// TwinCAT 3 PLC project Singleton1
// ProgramVersion: 3.1.4023.0
// libraries:
//   Tc2_Standard, * (Beckhoff Automation GmbH)
//   Tc2_System, * (Beckhoff Automation GmbH)
//   Tc3_Module, * (Beckhoff Automation GmbH)
//   VisuSymbols,3.5.10.0,System
// project tree:
//   / Class Diagram_2.TcCD (not stored), E_Color.TcDUT (not stored), GlobalTextList.TcGTLO, PlcTask.TcTTO (not stored), PLC_PRG.TcPOU, ProxyToSingleton.TcPOU, Proxy_Interface.TcIO (not stored), RealSingleton.TcPOU, Visualization Manager.TcVMO (not stored)
//   POUs/ MAIN.TcPOU (not stored)
//   VISUs/ Visualization.TcVIS
// real-time tasks:
//   TASK PlcTask: cycle T#10ms, priority 20, ADS port 350

// ---- PLC_PRG.TcPOU
PROGRAM PLC_PRG
VAR
	///Blue, highly opaque
	dwBlue: DWORD := 16#FF0000FF;
	///Green, highly opaque
	dwGreen: DWORD := 16#FF00FF00;
	///Yellow, highly opaque
	dwYellow: DWORD := 16#FFFFFFF0;
	///Creates 3 instances of the ProxyToSingleton class
	instance1: ProxyToSingleton;
	instance2: ProxyToSingleton;
	instance3: ProxyToSingleton;
	
	eInstance1 : E_Color;
	eInstance2 : E_Color;
	eInstance3 : E_Color;
	
END_VAR

//*************************************************************************************************************************************************************
//The PLC_PRG handles the instanciation of the possible background colours and the ProxyToSingleton instances in order to be used by the Visualization element.
//The viasualization element (The client) handles the request for background change on the RealSingleton object through the ProxyToSinlgeton instances.
//These request are first processed by the ProxyToSingleton object and then passed to the one and only RealSingleton instance.
//The default background colour of the RealSingleton object is 'Blue' 
//*************************************************************************************************************************************************************
// spanish
//PLC_PRG maneja la instanciación de los posibles colores de fondo y las instancias de ProxyToSingleton para ser utilizados por el elemento de visualización.
//El elemento de visualización (el cliente) maneja la solicitud de cambio de fondo en el objeto RealSingleton a través de las instancias de ProxyToSinlgeton.
//Estas solicitudes son procesadas primero por el objeto ProxyToSingleton y luego pasadas a la única instancia de RealSingleton.
//El color de fondo predeterminado del objeto RealSingleton es 'Azul'
//*************************************************************************************************************************************************************

CASE eInstance1 OF
	E_Color.Blue:
		instance1.Set_Background(dwBlue);
		eInstance1:=E_Color.NoColor;
	E_Color.Green:
		instance1.Set_Background(dwGreen);
		eInstance1:=E_Color.NoColor;
	E_Color.Yellow:
		instance1.Set_Background(dwYellow);
		eInstance1:=E_Color.NoColor;
END_CASE

CASE eInstance2 OF
	E_Color.Blue:
		instance2.Set_Background(dwBlue);
		eInstance2:=E_Color.NoColor;	
	E_Color.Green:
		instance2.Set_Background(dwGreen);
		eInstance2:=E_Color.NoColor;	
	E_Color.Yellow:
		instance2.Set_Background(dwYellow);
		eInstance2:=E_Color.NoColor;	
END_CASE

CASE eInstance3 OF
	E_Color.Blue:
		instance3.Set_Background(dwBlue);
		eInstance3:=E_Color.NoColor;	
	E_Color.Green:
		instance3.Set_Background(dwGreen);
		eInstance3:=E_Color.NoColor;	
	E_Color.Yellow:
		instance3.Set_Background(dwYellow);
		eInstance3:=E_Color.NoColor;	
END_CASE

END_PROGRAM

// ---- ProxyToSingleton.TcPOU
///This class is called ProxyToSingleton because it works as a Proxy of the Singleton class. It handles the creation and instanciation of the 
/// RealSingleton class. Something like the proper static method GetInstance(); in any singleton pattern.
///So the ProxyToSingleton class has a static Singleton object as a field and whenever we instanciate a 
/// ProxyToSingleton object we will have the RealSingleton object as its static field .realSingleton^
{attribute 'enable_dynamic_creation' := ''}
FUNCTION_BLOCK ProxyToSingleton IMPLEMENTS Proxy_Interface
VAR_STAT
	///Boolean value to check if there is already a Singleton instance
	bFirstInstance: BOOL := FALSE;
	///Pointer to the first and only instance of the Singleton class
	realSingleton: POINTER TO RealSingleton;
END_VAR

METHOD fb_init
VAR_INPUT
	/// TRUE: the Retain-variables are initialized (reset warm / reset cold)
	bInitRetains: BOOL;
	/// TRUE  the instance will be copied to the copy-code afterward (online change)
	bInCopyCode: BOOL;
END_VAR
//THIS FUNCTION WORKS AS THE CONSTRUCTOR OF THE ProxyToSingleton CLASS
// It handles the creation of the only RealSingleton object. It uses the concept of lazy instanciation.

//If the static property .bFirstInstance is TRUE
IF THIS^.bFirstInstance = TRUE
	
THEN
		//There is already a Singleton object.
		//So we don't have to do anything, this new ProxyToSingleton object will already have the address of the 
		// RealSingleton object in its pointer .realSingleton
	
	ELSE	//If the static property .bFirstInstance is FALSE
	
		//There is not a Singleton object so the ProxyToSingleton object calling the constructor 
		// should create the RealSingleton object in its pointer field .realSingleton 
		//Then we change the status of the static variable bFirstInstance to TRUE and avoid overwriting the realSingleton address.
		//If the Singleton object is destroyed, .bFirstInstance should be set to FALSE again.
		THIS^.bFirstInstance := TRUE;
		
		//Reference the value of the first RealSingleton instance to the FakeSingleton object to save 
		// the address of the real Singleton instance.
		THIS^.realSingleton := __NEW(RealSingleton);
END_IF
END_METHOD

///Illustrative method of the pattern
METHOD Set_Background
VAR_INPUT
	///HEX value to be set as background color
	newBackground: DWORD;
END_VAR
//The ProxyToSingleton object handles the request and send the appropiate reques to the one and only RealSingleton instance
THIS^.realSingleton^.Set_Background(newBackground);
END_METHOD

END_FUNCTION_BLOCK

// ---- RealSingleton.TcPOU
///This class is called RealSingleton because it works as singleton.  
///As long as we only instanciate ProxyToSingleton objects, this class will work as a Singleton class should work.
///The global access point to this class is the field .realSingleton^ in every ProxyToSingleton object.
{attribute 'enable_dynamic_creation' := ''}
FUNCTION_BLOCK RealSingleton IMPLEMENTS Proxy_Interface
VAR
	///Illustrative field of the pattern to store the HEX value for the background colour
	backgroundColour: DWORD;
END_VAR

METHOD fb_init
VAR_INPUT
	/// TRUE: the Retain-variables are initialized (reset warm / reset cold)
	bInitRetains: BOOL;
	/// TRUE  the instance will be copied to the copy-code afterward (online change)
	bInCopyCode: BOOL;
END_VAR
//The default valur for the background is set
THIS^.Set_Background(PLC_PRG.dwBlue);
END_METHOD

///Illustrative method of the pattern
METHOD Set_Background
VAR_INPUT
	///HEX value to be set as background color
	newBackground: DWORD;
END_VAR
//Writes the backgroundColour field to the passed newBackground value
THIS^.backgroundColour := newBackground;
END_METHOD

END_FUNCTION_BLOCK

// ---- GlobalTextList.TcGTLO
TEXTLIST GlobalTextList
  630 = "//The PLC_PRG handles the instanciation of the possible background colours and the ProxyToSingleton instances in order to be used by the Visualization element.\n//The viasualization element (The client) handles the request for background change on the RealSingleton object through the ProxyToSinlgeton instances.\n//These request are first processed by the ProxyToSingleton object and then passed to the one and only RealSingleton instance.\n//The default background colour of the RealSingleton object is 'Blue' "
  622 = "//The PLC_PRG handles the instanciation of the possible background colours and the ProxyToSingleton instances in order to be used by the Visualization element.\n//The visualization element (The client) handles the request for background change on the RealSingleton object through the ProxyToSinlgeton instances.\n//These request are first processed by the ProxyToSingleton object and then passed to the one and only RealSingleton instance.\n//The default background colour of the RealSingleton object is 'Blue' "
  596 = 'instance1.realSingleton^.\nbackgroundColor'
  621 = 'instance1.Set_Background(HEX color)'
  436 = 'instance2.realSingleton^.\nbackgroundColor'
  534 = 'instance2.Set_Background(HEX color)'
  774 = 'instance3.realSingleton^.\nbackgroundColor'
  50 = 'instance3.Set_Background(HEX color)'
  430 = 'The PLC_PRG handles the instanciation of the possible background colours and the ProxyToSingleton instances in order to be used by the Visualization element.\n'
END_TEXTLIST

// ---- VISUs/Visualization.TcVIS
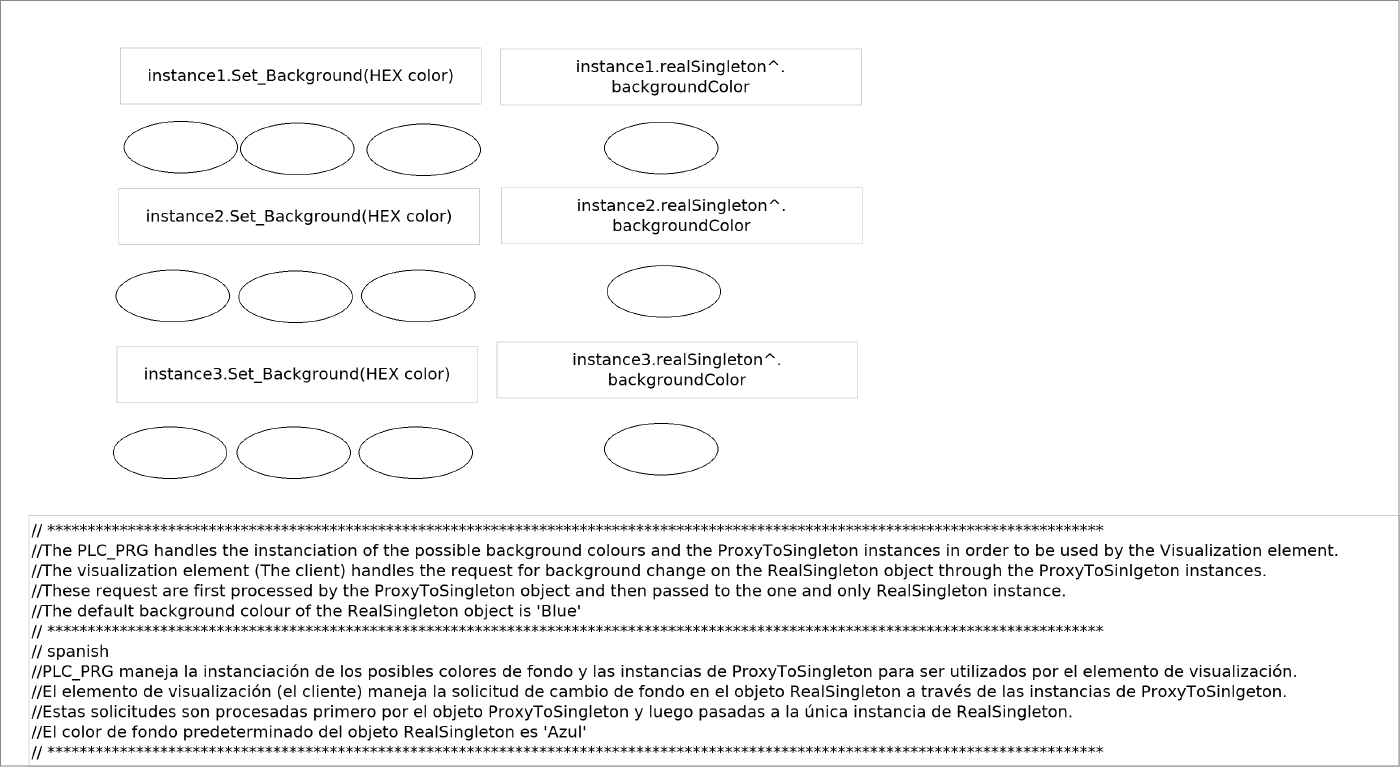
VISUALIZATION Visualization  // 1562x856
    Textfield (134,53 403x63), "instance1.Set_Background(HEX color)"
    Textfield (558,54 403x63), "instance1.realSingleton^. backgroundColor"
    Textfield (132,210 403x63), "instance2.Set_Background(HEX color)"
    Textfield (130,386 403x63), "instance3.Set_Background(HEX color)"
    Textfield (559,209 403x63), "instance2.realSingleton^. backgroundColor"
    Textfield (554,381 403x63), "instance3.realSingleton^. backgroundColor"
    Ellipse (138,135 127x58), colour variable: PLC_PRG.dwBlue
        OnMouseClick: execute {
            //PLC_PRG.instance1.Set_Background(newBackground:=PLC_PRG.dwBlue);
            PLC_PRG.eInstance1 := E_Color.Blue;
        }
    Ellipse (409,138 127x58), colour variable: PLC_PRG.dwYellow
        OnMouseClick: execute {
            //PLC_PRG.instance1.Set_Background(newBackground:=PLC_PRG.dwYellow);
            PLC_PRG.eInstance1 := E_Color.Yellow;
        }
    Ellipse (268,137 127x58), colour variable: PLC_PRG.dwGreen
        OnMouseClick: execute {
            //PLC_PRG.instance1.Set_Background(newBackground:=PLC_PRG.dwGreen);
            PLC_PRG.eInstance1 := E_Color.Green;
        }
    Ellipse (129,301 127x58), colour variable: PLC_PRG.dwBlue
        OnMouseClick: execute {
            //PLC_PRG.instance2.Set_Background(PLC_PRG.dwBlue);
            PLC_PRG.eInstance2 := E_Color.Blue;
        }
    Ellipse (403,301 127x58), colour variable: PLC_PRG.dwYellow
        OnMouseClick: execute {
            //PLC_PRG.instance2.Set_Background(PLC_PRG.dwYellow);
            PLC_PRG.eInstance2 := E_Color.Yellow;
        }
    Ellipse (266,302 127x58), colour variable: PLC_PRG.dwGreen
        OnMouseClick: execute {
            //PLC_PRG.instance2.Set_Background(PLC_PRG.dwGreen);
            PLC_PRG.eInstance2 := E_Color.Green;
        }
    Ellipse (126,476 127x58), colour variable: PLC_PRG.dwBlue
        OnMouseClick: execute {
            //PLC_PRG.instance3.Set_Background(PLC_PRG.dwBlue);
            PLC_PRG.eInstance3 := E_Color.Blue;
        }
    Ellipse (400,476 127x58), colour variable: PLC_PRG.dwYellow
        OnMouseClick: execute {
            //PLC_PRG.instance3.Set_Background(PLC_PRG.dwYellow);
            PLC_PRG.eInstance3 := E_Color.Yellow;
        }
    Ellipse (264,476 127x58), colour variable: PLC_PRG.dwGreen
        OnMouseClick: execute {
            //PLC_PRG.instance3.Set_Background(PLC_PRG.dwGreen);
            PLC_PRG.eInstance3 := E_Color.Green;
        }
    Ellipse (674,472 127x58), colour variable: PLC_PRG.instance3.realSingleton^.backgroundColour
    Ellipse (677,296 127x58), colour variable: PLC_PRG.instance2.realSingleton^.backgroundColour
    Ellipse (674,136 127x58), colour variable: PLC_PRG.instance1.realSingleton^.backgroundColour
    Textfield (32,575 1530x281), "// *********************************************************************************************************************************** //The PLC_PRG handles the instanciation of the possible background colours and the ProxyToSingleton instances in order to be used by the Visualization element. //The visualization element (The client) handles the request for background change on the RealSingleton object through the ProxyToSinlgeton instances. //These request are first processed by the ProxyToSingleton object and then passed to the one and only RealSingleton instance. //The default background colour of the RealSingleton object is 'Blue' // *********************************************************************************************************************************** // spanish //PLC_PRG maneja la instanciación de los posibles colores de fondo y las instancias de ProxyToSingleton para ser utilizados por el elemento de visualización. //El elemento de visualización (el cliente) maneja la solicitud de cambio de fondo en el objeto RealSingleton a través de las instancias de ProxyToSinlgeton. //Estas solicitudes son procesadas primero por el objeto ProxyToSingleton y luego pasadas a la única instancia de RealSingleton. //El color de fondo predeterminado del objeto RealSingleton es 'Azul' // ***********************************************************************************************************************************"
END_VISUALIZATION
